FUNCTION_BLOCK ADD_DINT (* IEC 61131-3 DINT Addition *)
  (* Standard: 61131-3 *)
  (* Version 0.0, 2004-12-15, JHC, Rockwell Automation, Converted from SRC format. *)
  (* Compiler header: package fb.rt.plc.math; *)
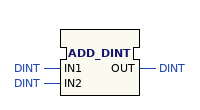
  VAR_INPUT
    IN1 : DINT; (* Augend *)
    IN2 : DINT; (* Addend *)
  END_VAR
  VAR_OUTPUT
    OUT : DINT; (* Sum *)
  END_VAR
END_FUNCTION_BLOCK
